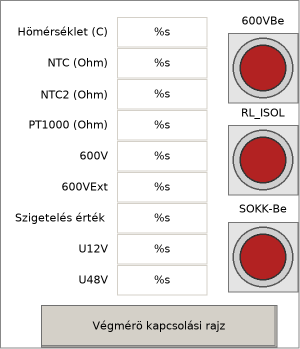
VISUALIZATION Vegmero_kezi  // 300x349
    PushSwitch (228,125 70x70), variable: VEGMERO.bRL_ISOL, behaviour: TOGGLE, style: Switch-PushSwitch-Red
    Label (233,103 60x20), "RL_ISOL"
    Textfield (117,141 90x30), "%s", text variable: VEGMERO.U600V_TRANS
    Textfield (117,48 90x30), "%s", text variable: VEGMERO.NTRES_CALC
    Textfield (117,110 90x30), "%s", text variable: VEGMERO.PTRES_CALC
    Label (11,48 100x30), "NTC (Ohm)"
    Label (11,110 100x30), "PT1000 (Ohm)"
    Label (11,141 100x30), "600V"
    PushSwitch (228,33 70x70), variable: VEGMERO.b600VBe, behaviour: TOGGLE, style: Switch-PushSwitch-Red
    Label (233,11 60x20), "600VBe"
    Textfield (117,265 90x30), "%s", text variable: VEGMERO.U48V_CAL
    Label (11,265 100x30), "U48V"
    Textfield (117,172 90x30), "%s", text variable: VEGMERO.U600VExt_TRANS
    Label (11,172 100x30), "600VExt"
    Textfield (117,203 90x30), "%s", text variable: VEGMERO.UISOL_TRANS
    Label (11,203 97x30), "Szigetelés érték"
    PushSwitch (228,222 70x70), variable: VEGMERO.PT_SOKK48V, behaviour: TOGGLE, style: Switch-PushSwitch-Red
    Label (233,199 60x20), "SOKK-Be"
    Textfield (117,234 90x30), "%s", text variable: VEGMERO.U12V_CAL
    Label (11,234 100x30), "U12V"
    Textfield (117,17 90x30), "%s", text variable: VEGMERO.rHoerzekelo_TRANS
    Label (11,17 100x30), "Hömérséklet (C)"
    Button (41,305 236x42), "Végmérö kapcsolási rajz", tooltip "Ultimate script-ben megírt parancsok pdf-ben", pressed state: Laser.bStartUltimate
        OnMouseUp: execute { VEGMERO.bStartSchematic:=TRUE; }
    Textfield (117,79 90x30), "%s", text variable: VEGMERO.NTRES2_CALC
    Label (11,80 100x30), "NTC2 (Ohm)"
END_VISUALIZATION

(* stored: Version 1.1.0.1, ProductVersion 3.1.4024.11
   Visu Vegmero_kezi: Id {2242c424-6e60-43e6-a796-bbb015cff537} *)
